# B&R Automation Studio project ManitouIHM_AS111
Automation Studio 4.9

## Configuration Config1

CPU 4PP045.0571-062, AutomationRuntime H3.10, Build 4.1.2, Vc V4.72.2

### Task classes (Cpu.sw)
```
Cyclic#1:
  TrameRecu <- TrameRecu.prg
  CanQueue <- SamplesCAN_Lib.LibCAN_Lib1_ST.CanQueue.prg
  Simulation <- Simulation.prg
VcDataObjects: Visu <- Visu.dob
Binaries: vccbar, vcpk, vcfntttf, vcctext, arial, vccdt, vcmgr, vccbtn, vcdsint, vcpdsw, vcptpp45, vctcal, vcshared, vccovl, vcfile, vcpdpp45, vcgclass, arialbd, vcrt, Visu02, Visu03, udbdef, Visu01, vcclbox, vcdsloc, vccbmp, vcbclass, vcalarm, vcpfpp45, vccnum, vccstr, vccshape, iomap, asfw, sysconf, arconfig, ashwd, ashwac
Libraries: CAN_Lib, vcresman, astime, asieccon, fileio, dataobj, runtime
```

### Hardware
```
4PP045_0571_062 : 4PP045.0571-062 v1.0.5.0
  Connector IF1:
    ActivateDevice = 1
    Mode = Manual
    InternetAddress = 10.16.7.83
    SubnetMask = 255.255.0.0
  VcObjectName = Visu
  KeyMappingFile = VC\4PP045_0571_062.dis
4PP045_IF23-1 : 4PP045.IF23-1 v1.0.0.0  [SS -> 4PP045_0571_062.SS1]
  Connector IF3:
    Baudrate = 250000
    IdentifierLength = 1
    ReceiveTimeout = 20
    ActivateCanOpen = 1
    p100c_parametervalue = 1000
    p100d_parametervalue = 3
```

## Logical view

Binary libraries used (declarations not repeated): CAN_Lib

### Global.typ - Global data types
```iecst
TYPE
	Trame : 	STRUCT
		CanDevice1 : STRING[80];
		Frame : INFO_typ;
		Info : CANread;
		New_Member : USINT;
	END_STRUCT;
END_TYPE
```

### Global.var - Global variables
```iecst
VAR
	SPU_TX_LED_03 : USINT;
	LV_FreinAMain : USINT; (*Frein à main icone*)
	SPU_TX_LCD_04 : USINT; (*ICON LCD 000 = Neutral, 001=Forward, 010 = Reverse, 011 = Off, 111 = HW input*)
	LV_Batterie : USINT; (*Batterie*)
	SPU_TX_LED_04 : USINT; (*Batterie icone*)
	SPU_TX_LED_01 : USINT := 1; (*Ceinture icone*)
	LV_Pression_huile : USINT; (*Pression huile*)
	LV_Huile_Moteur : USINT; (*Huile moteur*)
	LV_Tmp_Moteur : USINT; (*Temperature du moteur*)
	LV_Ceinture : USINT; (*Ceinture*)
	Octet : ARRAY[0..7] OF USINT;
END_VAR
```

- Visualisation Logical/Visu (not shown)

### Program Logical/TrameRecu (IEC)

#### Variables.var
```iecst
VAR
	BlinkTimer : TIME := T#1s;
	i : USINT;
	k : USINT;
	CANreader : ARRAY[0..2] OF Trame;
	Octet1 : USINT;
	Octet2 : USINT;
	Octet3 : USINT;
	Octet4 : USINT;
	Octet5 : USINT;
	Octet6 : USINT;
	Octet7 : USINT;
	Octet8 : USINT;
END_VAR
```

#### Main.st
```iecst
PROGRAM _INIT
	// Trame du SPU

	CANreader[0].Info.can_id := 16#18FF1021; //SPU_HMI_TRAME1
	CANreader[1].Info.can_id := 16#18FF2021; //SPU_HMI_TRAME2
	CANreader[2].Info.can_id := 16#18FF3021; //SPU_HMI_TRAME3

	FOR k:= 0 TO 2 DO
		CANreader[k].ConfigComm.enable := TRUE;
		CANreader[k].ConfigComm.baud_rate := 250;
	END_FOR;

END_PROGRAM

PROGRAM _CYCLIC

	//lire la trame recue sur le bus CAN

	FOR k := 0 TO 2 DO
		CANreader[k].Frame.received;
	END_FOR

	//Acquisition des octets et mettre dans les variables correspondantes

	FOR k := 0 TO 7 DO

	END_FOR

	// met les octets dans les variables USINT correspondante pour que je peux les retranscrire sur la page maintenance

	Octet1 := Octet[0];
	Octet2 := Octet[1];
	Octet3 := Octet[2];
	Octet4 := Octet[3];
	Octet5 := Octet[4];
	Octet6 := Octet[5];
	Octet7 := Octet[6];
	Octet8 := Octet[7];

	// Si Trame SPU_TX_LED_01 = 1 alors allumé le voyant ceinture sinon éteindre

	IF SPU_TX_LED_01 = 1 THEN
		LV_Ceinture := 1;
	ELSE
		LV_Ceinture := 0;
	END_IF

	// Si Trame SPU_TX_LED_03 = 1 alors allumé le voyant Frein à main sinon éteindre

	IF SPU_TX_LED_03 = 1 THEN
		LV_FreinAMain := 1;
	ELSE
		LV_FreinAMain := 0;
	END_IF

	// Si Trame SPU_TX_LED_016 = 1 alors allumé le voyant batterie sinon éteindre

	IF SPU_TX_LED_04 = 1 THEN
		LV_Batterie := 1 ;
	ELSIF SPU_TX_LED_04 = 0 THEN
		LV_Batterie := 0 ;
	END_IF

END_PROGRAM

PROGRAM _EXIT

END_PROGRAM
```

### Program Logical/Simulation (IEC)

#### Variables.var
```iecst
VAR
	Hauteur : USINT;
	Essence : USINT;
	Vitesse : USINT;
END_VAR
```

#### Main.st
```iecst
PROGRAM _INIT
	(* Insert code here *)
	Vitesse := 11;
	Hauteur := 4;
	Essence := 50;
END_PROGRAM

PROGRAM _CYCLIC
	(* Insert code here *)

END_PROGRAM

PROGRAM _EXIT
	(* Insert code here *)

END_PROGRAM
```


### Package Logical/SamplesCAN_Lib/LibCAN_Lib1_ST - CANopen, CANqueue, CANrd, CANquwr, CANinfo

### Program Logical/SamplesCAN_Lib/LibCAN_Lib1_ST/CanQueue (IEC)

#### CanQueue.st - CANopen, CANqueue, CANrd, CANquwr, CANinfo
```iecst
PROGRAM	_INIT
	(* Initialize Names	and	ID's for the send program *)
	(* The device name for the CAN send	bus. One can find the name in the Physical View -> PLC Address. *)

	canQueueReadWrite.CANopen_0.enable := TRUE;
	canQueueReadWrite.CANopen_0.device := ADR('SS1.IF1 /BD=500000 /EX=0');
	canQueueReadWrite.CANopen_0.cob_anz := 100;
	canQueueReadWrite.CANopen_0.error_adr := ADR(canQueueReadWrite.canError_0);
	canQueueReadWrite.CANopen_0();

	canQueueReadWrite.CANopen_1.enable := TRUE;
	canQueueReadWrite.CANopen_1.device := ADR('SS1.IF2 /BD=500000 /EX=0');
	canQueueReadWrite.CANopen_1.cob_anz := 100;
	canQueueReadWrite.CANopen_1.error_adr := ADR (canQueueReadWrite.canError_1);
	canQueueReadWrite.CANopen_1();

END_PROGRAM

PROGRAM	_CYCLIC

	canQueueReadWrite.CANinfo_0();
	canQueueReadWrite.CANinfo_1();

	CASE canQueueReadWrite.step OF

		STEP_INIT:
			IF canQueueReadWrite.CANopen_1.status = 0 AND canQueueReadWrite.CANopen_0.status = 0 THEN
				canQueueReadWrite.CANinfo_0.enable := TRUE;
				canQueueReadWrite.CANinfo_0.info_adr := ADR(canQueueReadWrite.canInfo_0);
				canQueueReadWrite.CANinfo_0.us_ident := canQueueReadWrite.CANopen_0.us_ident;

				canQueueReadWrite.CANinfo_1.enable := TRUE;
				canQueueReadWrite.CANinfo_1.info_adr := ADR(canQueueReadWrite.canInfo_1);
				canQueueReadWrite.CANinfo_1.us_ident := canQueueReadWrite.CANopen_1.us_ident;

				canQueueReadWrite.step := STEP_DEFINE_QUEUE;
			END_IF

		STEP_DEFINE_QUEUE:
			canQueueReadWrite.CANqueue_1.enable := TRUE;
			canQueueReadWrite.CANqueue_1.us_ident := canQueueReadWrite.CANopen_1.us_ident;
			canQueueReadWrite.CANqueue_1.can_id := MY_CAN_IDENTIFIER;
			canQueueReadWrite.CANqueue_1.size := 100;
			canQueueReadWrite.CANqueue_1();
			IF canQueueReadWrite.CANqueue_1.status = 0 THEN
				canQueueReadWrite.step := STEP_QUICKWRITE;
			END_IF

		STEP_QUICKWRITE:
			canQueueReadWrite.CANquwr_0.enable := TRUE;
			canQueueReadWrite.CANquwr_0.us_ident := canQueueReadWrite.CANopen_0.us_ident;
			canQueueReadWrite.CANquwr_0.can_id := MY_CAN_IDENTIFIER;
			canQueueReadWrite.CANquwr_0.data_adr := ADR(canQueueReadWrite.writeData);
			canQueueReadWrite.CANquwr_0.data_lng := SIZEOF (canQueueReadWrite.writeData);

			FOR n:=0 TO MAX_SEND_FRAMES DO
				canQueueReadWrite.CANquwr_0();
				IF canQueueReadWrite.CANquwr_0.status = 0 THEN
					canQueueReadWrite.successWrite := canQueueReadWrite.successWrite + 1;
					canQueueReadWrite.writeData[0] := canQueueReadWrite.successWrite;
				ELSIF canQueueReadWrite.CANquwr_0.status <> canERR_CAN_QFULL THEN
					canQueueReadWrite.step := STEP_ERROR;
					EXIT;
				END_IF
			END_FOR
			canQueueReadWrite.step := STEP_READ_QUEUE;

		STEP_READ_QUEUE:
			canQueueReadWrite.CANrd_1.enable := TRUE;
			canQueueReadWrite.CANrd_1.q_ident := canQueueReadWrite.CANqueue_1.q_ident;
			canQueueReadWrite.CANrd_1.data_adr := ADR(canQueueReadWrite.readData);
			canQueueReadWrite.CANrd_1();
			WHILE canQueueReadWrite.CANrd_1.status = 0 DO
				canQueueReadWrite.successRead := canQueueReadWrite.successRead + 1;
				canQueueReadWrite.writeData[1] := canQueueReadWrite.successRead;
				canQueueReadWrite.CANrd_1();
			END_WHILE;

			canQueueReadWrite.step := STEP_QUICKWRITE;

		STEP_ERROR:	(* Error Handling *)
	END_CASE
END_PROGRAM

PROGRAM	_EXIT
END_PROGRAM
```

#### CanQueue.typ - Local data types
```iecst
TYPE
	CanQueue_Steps :
		(
		STEP_ERROR := 255,
		STEP_INIT := 1,
		STEP_DEFINE_QUEUE := 2,
		STEP_QUICKWRITE := 3,
		STEP_READ_QUEUE := 4
		);
	CanQueueReadWrite_typ : 	STRUCT
		step : CanQueue_Steps := STEP_INIT;
		canDevice0 : STRING[80];
		canDevice1 : STRING[80];
		writeData : ARRAY[0..1]OF UDINT;
		readData : ARRAY[0..1]OF UDINT;
		CANopen_0 : CANopen;
		CANopen_1 : CANopen;
		CANquwr_0 : CANquwr;
		CANqueue_1 : CANqueue;
		CANrd_1 : CANrd;
		CANinfo_0 : CANinfo;
		CANinfo_1 : CANinfo;
		successRead : UDINT;
		successWrite : UDINT;
		errorCount : UINT;
		stopTest : BOOL := FALSE;
		canError_1 : UINT;
		canError_0 : UINT;
		canInfo_1 : INFO_typ;
		canInfo_0 : INFO_typ;
	END_STRUCT;
END_TYPE
```

#### CanQueue.var - Local variables
```iecst
VAR CONSTANT
	MAX_SEND_FRAMES : USINT := 10;
	MY_CAN_IDENTIFIER : UDINT := 257;
END_VAR
VAR
	canQueueReadWrite : CanQueueReadWrite_typ;
	n : USINT;
END_VAR
```
